// TIA Portal V16 export
// export: Created 2021-07-12T14:47:18.9125014Z, ExportSetting WithDefaults, DisplayName Totally Integrated Automation Portal, DisplayVersion V16, DisplayName TIA Portal Version Control Interface, DisplayVersion V16, DisplayName TIA Portal Openness, DisplayVersion V16, DisplayName STEP 7 Professional, DisplayVersion V16, DisplayName STEP 7 Safety, DisplayVersion V16, DisplayName WinCC Professional, DisplayVersion V16
TYPE "LSimaHydTO_typeInternalCmdTracking"
TITLE = LSimaHydTO_typeInternalCmdTracking
// Command tracking
// stored: IsFailsafeCompliant false
   STRUCT
      CommandID : UDInt := 0;   // Command ID for tracking
      State : Word := 0;   // Command state
   END_STRUCT;
END_TYPE
